TYPE VEC3 :
STRUCT
	x: REAL;
	y: REAL;
	z: REAL;
END_STRUCT
END_TYPE

(* stored: Version 1.1.0.1, ProductVersion 3.1.0.25
   DUT VEC3: Id {5162ec0b-682f-43ed-8de7-55d89508de83} *)
